FUNCTION_BLOCK FB_Absolute_Example
VAR_INPUT
	bEnable		:BOOL;
	fPosition1	:LREAL;
	fPosition2	:LREAL;
	fPosition3	:LREAL;
	tDelay		:TIME;	
	fVelocity	:LREAL;
	
END_VAR
VAR_OUTPUT
	bError		:BOOL;
	sStatus		:STRING;
END_VAR

VAR
	fb_Power		: MC_Power;
	stateDataFlow	: (RESET_STATE, FIRST_MOVE_STATE, FIRST_MOTION_CONTROL_STATE, FIRST_WAIT_STATE, 
SECOND_MOVE_STATE, SECOND_MOTION_CONTROL_STATE, SECOND_WAIT_STATE, THIRD_MOVE_STATE,THIRD_MOTION_CONTROL_STATE,THIRD_WAIT_STATE, ERROR_STATE):=RESET_STATE;
	fbTimer			:TON;	
	fb_MoveAbsolute: MC_MoveAbsolute;
END_VAR
VAR_IN_OUT
	Axis :		AXIS_REF;
END_VAR


fbTimer(PT:=tDelay);

CASE stateDataFlow OF
	
RESET_STATE:
		bError			:=FALSE;
		sStatus			:='Beklemede';
		
		IF bEnable THEN
			stateDataFlow:=FIRST_MOVE_STATE;
			ELSIF NOT Axis.Status.Operational THEN
				stateDataFlow:=ERROR_STATE;
				sStatus:='Enable değil';
		END_IF
	fb_Power(
	Axis:= Axis, 
	Enable:=bEnable , 
	Enable_Positive:= bEnable, 
	Enable_Negative:=bEnable , 
	Override:=100 ,);
	

FIRST_MOVE_STATE:
	
	fb_MoveAbsolute.Position:=fPosition1;
	fb_MoveAbsolute.Execute 	:= TRUE;
	IF Axis.Status.Moving THEN 
		stateDataFlow:=FIRST_MOTION_CONTROL_STATE;
		sStatus:= '1. Noktaya gidiyor';
		ELSIF Axis.Status.Error OR fb_MoveAbsolute.Error THEN
		
		sStatus		:='1. noktaya giderken hataya geçti'	;
		stateDataFlow:=ERROR_STATE;
		
	END_IF 
	
FIRST_MOTION_CONTROL_STATE:
	IF fb_MoveAbsolute.Done THEN 
			stateDataFlow:=FIRST_WAIT_STATE;
			fb_MoveAbsolute.Execute:=FALSE;
		END_IF
	
FIRST_WAIT_STATE:

		fbTimer.IN:=TRUE;
		sStatus		:='1. noktada bekliyor ';
		
		IF fbTimer.Q THEN 
			fbTimer.IN:=FALSE;
			stateDataFlow:=SECOND_MOVE_STATE;
		END_IF	
		
SECOND_MOVE_STATE	:

	fb_MoveAbsolute.Position:=fPosition2;
	fVelocity:=fVelocity/2;
			fb_MoveAbsolute.Execute 	:= TRUE;
			IF Axis.Status.Moving THEN 
				
				stateDataFlow:=SECOND_MOTION_CONTROL_STATE;
				sStatus:= '2. Noktaya gidiyor';
				ELSIF Axis.Status.Error OR fb_MoveAbsolute.Error THEN
				
				sStatus		:='2. noktaya giderken hataya geçti';
				stateDataFlow:=ERROR_STATE;
			END_IF

SECOND_MOTION_CONTROL_STATE:
			
		IF fb_MoveAbsolute.Done THEN
			stateDataFlow := SECOND_WAIT_STATE;
			fb_MoveAbsolute.Execute:=FALSE;
			 
		END_IF
		
SECOND_WAIT_STATE:
	fbTimer.IN:=TRUE;
		
		sStatus		:='2. noktada bekliyor ';
		
		IF fbTimer.Q THEN 
			fbTimer.IN:=FALSE;
			stateDataFlow:=THIRD_MOVE_STATE;
		END_IF

		
		
		
THIRD_MOVE_STATE	:	

	fb_MoveAbsolute.Position:=fposition3;
	
			fb_MoveAbsolute.Execute 	:= TRUE;
			IF Axis.Status.Moving THEN 
				
				stateDataFlow:=THIRD_MOTION_CONTROL_STATE;
				sStatus:= '3. Noktaya gidiyor';
				ELSIF Axis.Status.Error OR fb_MoveAbsolute.Error THEN
				
				sStatus		:='3. noktaya giderken hataya geçti';
				stateDataFlow:=ERROR_STATE;
			END_IF

			
THIRD_MOTION_CONTROL_STATE:
	
	IF fb_MoveAbsolute.Done THEN
			stateDataFlow := THIRD_WAIT_STATE;
			fb_MoveAbsolute.Execute:=FALSE;
			 
		END_IF

				
THIRD_WAIT_STATE:
	fbTimer.IN:=TRUE;
		sStatus		:='3. noktada bekliyor ';
		
		IF fbTimer.Q THEN 
			fbTimer.IN:=FALSE;
			stateDataFlow:=RESET_STATE;
		END_IF

		
ERROR_STATE:
	bError :=FALSE;
		
		IF NOT bEnable THEN
			fbTimer(IN:= FALSE);
			stateDataFlow:=RESET_STATE;
		END_IF

	END_CASE

fb_MoveAbsolute(
	Axis:= Axis, 
	Velocity:=fVelocity ,);
	Axis.ReadStatus();

END_FUNCTION_BLOCK

(* stored: Version 1.1.0.1, ProductVersion 3.1.4024.12
   POU FB_Absolute_Example: Id {f486185f-5703-4886-844e-fd9f963ca55d}, SpecialFunc None *)
